// TIA Portal V20 export
VAR_GLOBAL   // PLC tag table "VALVE_TYPES"
END_VAR
VAR_GLOBAL CONSTANT   // user constants
   Ball : Int := 1;   // Ball valve (on/off, fast actuation)
   Butterfly : Int := 2;   // Butterfly valve (throttling, low pressure drop)
   Diaphragm : Int := 3;   // Diaphragm valve (hygienic / corrosive media)
   Globe : Int := 4;   // Globe valve (precise throttling, high pressure drop)
   Needle : Int := 5;   // Needle valve (very fine throttling, low flow)
END_VAR
